% RSLogix 500 project ANDORNOTCLR.RSS, saved by version 9.00.00.04 %
PROJECT "UNTITLED"    % processor: Bul.1763 MicroLogix 1100 Series B %

PROGRAM FILES
  LAD 2   7 rungs

DATA FILES
  O0 OUTPUT  4 elements
  I1 INPUT  6 elements
  S2 STATUS  66 elements
  B3 BINARY  4 elements
  T4 TIMER  1 elements
  C5 COUNTER  1 elements
  R6 CONTROL  1 elements
  N7 INTEGER  1 elements
  F8 FLOAT  1 elements

LADDER 2
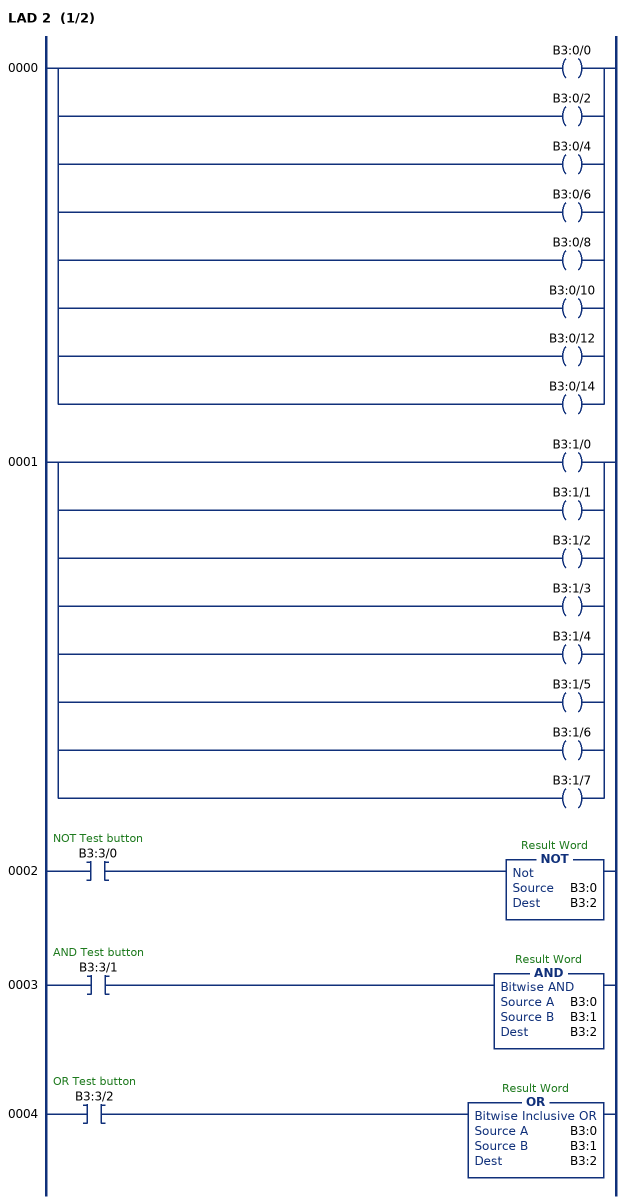
% Rung: 0 %
SOR BST OTE B3:0/0 NXB OTE B3:0/2 NXB OTE B3:0/4 NXB OTE B3:0/6 NXB OTE B3:0/8 NXB OTE B3:0/10 NXB OTE B3:0/12 NXB OTE B3:0/14 BND EOR
% Rung: 1 %
SOR BST OTE B3:1/0 NXB OTE B3:1/1 NXB OTE B3:1/2 NXB OTE B3:1/3 NXB OTE B3:1/4 NXB OTE B3:1/5 NXB OTE B3:1/6 NXB OTE B3:1/7 BND EOR
% Rung: 2 %
SOR XIC B3:3/0 NOT B3:0 B3:2 EOR
%   B3:3/0  "NOT Test button" %
%   B3:0  "Static Word 1" %
%   B3:2  "Result Word" %
% Rung: 3 %
SOR XIC B3:3/1 AND B3:0 B3:1 B3:2 EOR
%   B3:3/1  "AND Test button" %
%   B3:0  "Static Word 1" %
%   B3:1  "Static Word 2" %
%   B3:2  "Result Word" %
% Rung: 4 %
SOR XIC B3:3/2 OR B3:0 B3:1 B3:2 EOR
%   B3:3/2  "OR Test button" %
%   B3:0  "Static Word 1" %
%   B3:1  "Static Word 2" %
%   B3:2  "Result Word" %

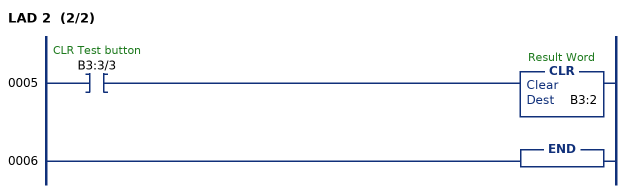
% Rung: 5 %
SOR XIC B3:3/3 CLR B3:2 EOR
%   B3:3/3  "CLR Test button" %
%   B3:2  "Result Word" %
% Rung: 6 %
SOR END EOR
